FUNCTION_BLOCK PAEChainConveyor EXTENDS PAETransport
VAR_INPUT
END_VAR
VAR_OUTPUT
END_VAR
VAR
END_VAR

END_FUNCTION_BLOCK

(* stored: Version 1.1.0.1, ProductVersion 3.1.4020.12
   POU PAEChainConveyor: Id {5f28b255-3cb9-49e0-975d-3e702a8ae4cd}, SpecialFunc None *)
